{attribute addProperty BoxType "EL3681-0000-0020"}
{attribute addProperty Id "StatusAT %I*Status_B1CD163B1621ValueAT %I*DINT32417"}
{attribute addProperty CRC "376365911"}
{attribute addProperty SizeInBites "48"}
{attribute addProperty SizeInBytes "6"}
TYPE SAI_Inputs_166EE357 :
STRUCT
	{attribute addProperty Name "Status"}
	Status AT %I* : Status_B1CD163B;
	{attribute addProperty Name "Value"}
	Value AT %I* : DINT;
END_STRUCT
END_TYPE

(* stored: Version 1.2.0.0, ProductVersion 3.1.4024.9
   DUT SAI_Inputs_166EE357: Id {fc401274-0305-4065-8d9b-8734d37fc5b0} *)
